TYPE EL3413_PM_OutputsAuxiliary :
STRUCT
	{attribute addProperty Name "Index"}
	Index AT %Q*: USINT;
	{attribute addProperty Name "Channel"}
	Channel AT %Q*: USINT;
END_STRUCT
END_TYPE

(* stored: Version 1.1.0.1, ProductVersion 3.1.4024.9
   DUT EL3413_PM_OutputsAuxiliary: Id {8213b8e1-5cce-0bd6-3785-ffa5caa76186} *)
